SYSTEM CONVEYORS (* System Configuration *)
  (* Standard: 61499-1 *)
  (* Version 0.4, 2009-03-05, JHC, Holobloc Inc., Deleted Application. *)
  (* Version 0.3, 2003-12-05, JHC, Rockwell Automation, Renamed from NEWSYSTEM. *)
  (* Version 0.2, 2002-11-05, JHC, Rockwell Automation, Fixed missing (empty) FBD in Application. *)
  (* Version 0.1, 2002-01-17, JHC, Rockwell Automation, Minor cleanup *)
  (* Version 0.0, 2000-05-27, JHC, Rockwell Automation *)
  DEVICE VIEW : FRAME_DEVICE(BOUNDS := [500,30,520,500])
    RESOURCE VIEW_Resource : VIEW_PANEL(DIA := 50, SIZE := [10,10])
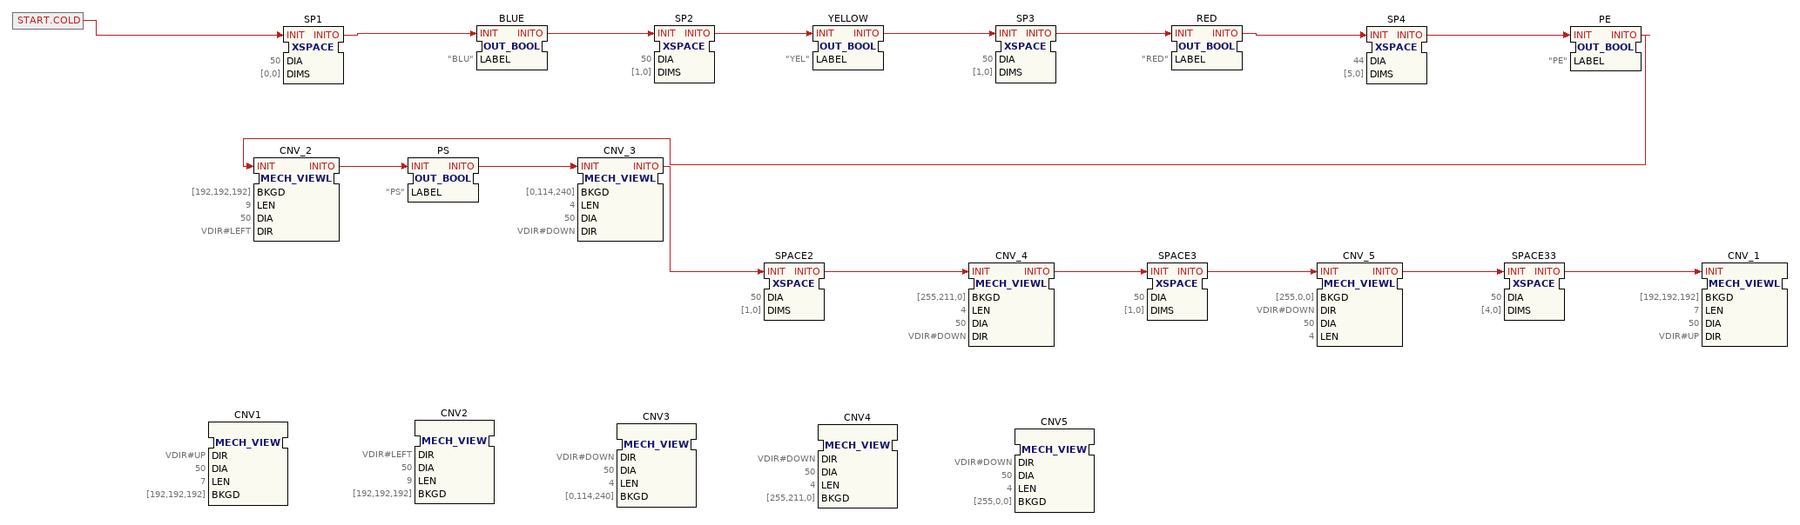
      FBS
        CNV1 : MECH_VIEW(DIR := VDIR#UP, DIA := 50, LEN := 7, BKGD := [192,192,192]);
        CNV2 : MECH_VIEW(DIR := VDIR#LEFT, DIA := 50, LEN := 9, BKGD := [192,192,192]);
        CNV3 : MECH_VIEW(DIR := VDIR#DOWN, DIA := 50, LEN := 4, BKGD := [0,114,240]);
        CNV4 : MECH_VIEW(DIR := VDIR#DOWN, DIA := 50, LEN := 4, BKGD := [255,211,0]);
        CNV5 : MECH_VIEW(DIR := VDIR#DOWN, DIA := 50, LEN := 4, BKGD := [255,0,0]);
        SPACE2 : XSPACE(DIA := 50, DIMS := [1,0]);
        SPACE3 : XSPACE(DIA := 50, DIMS := [1,0]);
        BLUE : OUT_BOOL(LABEL := "BLU");
        YELLOW : OUT_BOOL(LABEL := "YEL");
        RED : OUT_BOOL(LABEL := "RED");
        SP1 : XSPACE(DIA := 50, DIMS := [0,0]);
        SP2 : XSPACE(DIA := 50, DIMS := [1,0]);
        SP3 : XSPACE(DIA := 50, DIMS := [1,0]);
        SP4 : XSPACE(DIA := 44, DIMS := [5,0]);
        SPACE33 : XSPACE(DIA := 50, DIMS := [4,0]);
        PS : OUT_BOOL(LABEL := "PS");
        PE : OUT_BOOL(LABEL := "PE");
        CNV_2 : MECH_VIEWL(BKGD := [192,192,192], LEN := 9, DIA := 50, DIR := VDIR#LEFT);
        CNV_3 : MECH_VIEWL(BKGD := [0,114,240], LEN := 4, DIA := 50, DIR := VDIR#DOWN);
        CNV_4 : MECH_VIEWL(BKGD := [255,211,0], LEN := 4, DIA := 50, DIR := VDIR#DOWN);
        CNV_5 : MECH_VIEWL(BKGD := [255,0,0], DIR := VDIR#DOWN, DIA := 50, LEN := 4);
        CNV_1 : MECH_VIEWL(BKGD := [192,192,192], LEN := 7, DIA := 50, DIR := VDIR#UP);
      END_FBS
      EVENT_CONNECTIONS
        START.COLD TO SP1.INIT;
        SP1.INITO TO BLUE.INIT;
        BLUE.INITO TO SP2.INIT;
        SP2.INITO TO YELLOW.INIT;
        YELLOW.INITO TO SP3.INIT;
        SP3.INITO TO RED.INIT;
        RED.INITO TO SP4.INIT;
        SP4.INITO TO PE.INIT;
        PE.INITO TO CNV_2.INIT;
        CNV_2.INITO TO PS.INIT;
        PS.INITO TO CNV_3.INIT;
        CNV_3.INITO TO SPACE2.INIT;
        SPACE2.INITO TO CNV_4.INIT;
        CNV_4.INITO TO SPACE3.INIT;
        SPACE3.INITO TO CNV_5.INIT;
        CNV_5.INITO TO SPACE33.INIT;
        SPACE33.INITO TO CNV_1.INIT;
      END_CONNECTIONS
    END_RESOURCE
  END_DEVICE
  DEVICE HMI : FRAME_DEVICE(BOUNDS := [0,300,500,500])
    RESOURCE HMI_RESOURCE : VIEW_PANEL(DIA := 50, SIZE := [10,10])
    END_RESOURCE
  END_DEVICE
END_SYSTEM
